// TIA Portal project "OPTS_scale_main_V1" (V16)

(* hardware
DEVICE "S71500/ET200MP station_1"  S7-1500 station
   slot 0: "Rail_0"  Rack  6ES7 590-1***0-0AA0
   slot 1: "PLC_1"  CPU 1516F-3 PN/DP  6ES7 516-3FN01-0AB0  V1.8
      slot 3: "CPU display_1"  6ES7591-1BA00-0AA0
      slot 32768: "PROFINET interface_1"  X1
         slot 32769: "Port_1"  X1 P1
         slot 32770: "Port_2"  X1 P2
      slot 33024: "PROFINET interface_2"  X2
         slot 33025: "Port_1"  X2 P1
      slot 33280: "DP interface_1"  X3
   slot 2: "DI 32x24VDC HF_1"  DI 32x24VDC HF  6ES7 521-1BL00-0AB0  V2.1
   slot 3: "DQ 32x24VDC/0.5A ST_1"  DQ 32x24VDC/0.5A ST  6ES7 522-1BL00-0AB0  V2.0
   slot 4: "AI 8xU/I/RTD/TC ST_1"  AI 8xU/I/RTD/TC ST  6ES7 531-7KF00-0AB0  V2.0
   slot 5: "AQ 4xU/I ST_1"  AQ 4xU/I ST  6ES7 532-5HD00-0AB0  V2.0
DEVICE "HMI_1"  HMI.Device
*)

// ===== PLC "PLC_1"  CPU 1516F-3 PN/DP =====

VAR_GLOBAL   // PLC tag table "OPTS_tag_table"
   "onOffSwitch" AT %I2.0 : Bool;
   "FL_PositionSensor" AT %IW138 : Int;
   "FR_PositionSensor" AT %IW140 : Int;
   "BL_PositionSensor" AT %IW132 : Int;
   "BR_PositionSensor" AT %IW130 : Int;
   "sensorXValue" AT %IW134 : Int;
   "sensorZValue" AT %IW136 : Int;
   "flOut" AT %QW4 : Int;
   "frOut" AT %QW6 : Int;
END_VAR

DATA_BLOCK "SensorProcessing_DB"   // DB1
{ S7_Optimized_Access := 'TRUE' }
VERSION : 0.1
// stored: InstanceOfName SensorProcessing
"SensorProcessing"
BEGIN
END_DATA_BLOCK

DATA_BLOCK "TargetInDistance_DB"   // DB2
{ S7_Optimized_Access := 'TRUE' }
VERSION : 0.1
// stored: InstanceOfName TargetInDistance
"TargetInDistance"
BEGIN
END_DATA_BLOCK

DATA_BLOCK "TargetInDistance_DB_1"   // DB3
{ S7_Optimized_Access := 'TRUE' }
VERSION : 0.1
// stored: InstanceOfName TargetInDistance
"TargetInDistance"
BEGIN
END_DATA_BLOCK

DATA_BLOCK "TargetInDistance_DB_2"   // DB4
{ S7_Optimized_Access := 'TRUE' }
VERSION : 0.1
// stored: InstanceOfName TargetInDistance
"TargetInDistance"
BEGIN
END_DATA_BLOCK

DATA_BLOCK "TargetInDistance_DB_3"   // DB5
{ S7_Optimized_Access := 'TRUE' }
VERSION : 0.1
// stored: InstanceOfName TargetInDistance
"TargetInDistance"
BEGIN
END_DATA_BLOCK

FUNCTION_BLOCK "SensorProcessing"   // FB1, FBD
{ S7_Optimized_Access := 'TRUE' }
VERSION : 0.1
   VAR_INPUT
      sensorX : Int;
      sensorZ : Int;
      scale : Real;
      pi : Real;
      edgeToMiddle : Real := 150.0;
   END_VAR
   VAR_OUTPUT
      LA_FL_Target : Real;
      LA_FR_Target : Real;
      LA_BL_Target : Real;
      LA_BR_Target : Real;
   END_VAR
   VAR
      xActuatorAdjustVolt : Real;
      zActuatorAdjustVolt : Real;
      xActuatorAdjustVoltInv : Real;
      zActuatorAdjustVoltInv : Real;
   END_VAR
   VAR_TEMP
      xAngle : Real;
      zAngle : Real;
      xAngleTangent : Real;
      zAngleTangent : Real;
      xActuatorAdjust : Real;
      zActuatorAdjust : Real;
      xActuatorAdjustNorm : Real;
      zActuatorAdjustNorm : Real;
   END_VAR
BEGIN

REGION Network 1
   // Converting sensor data for X axis to an angle in radian.
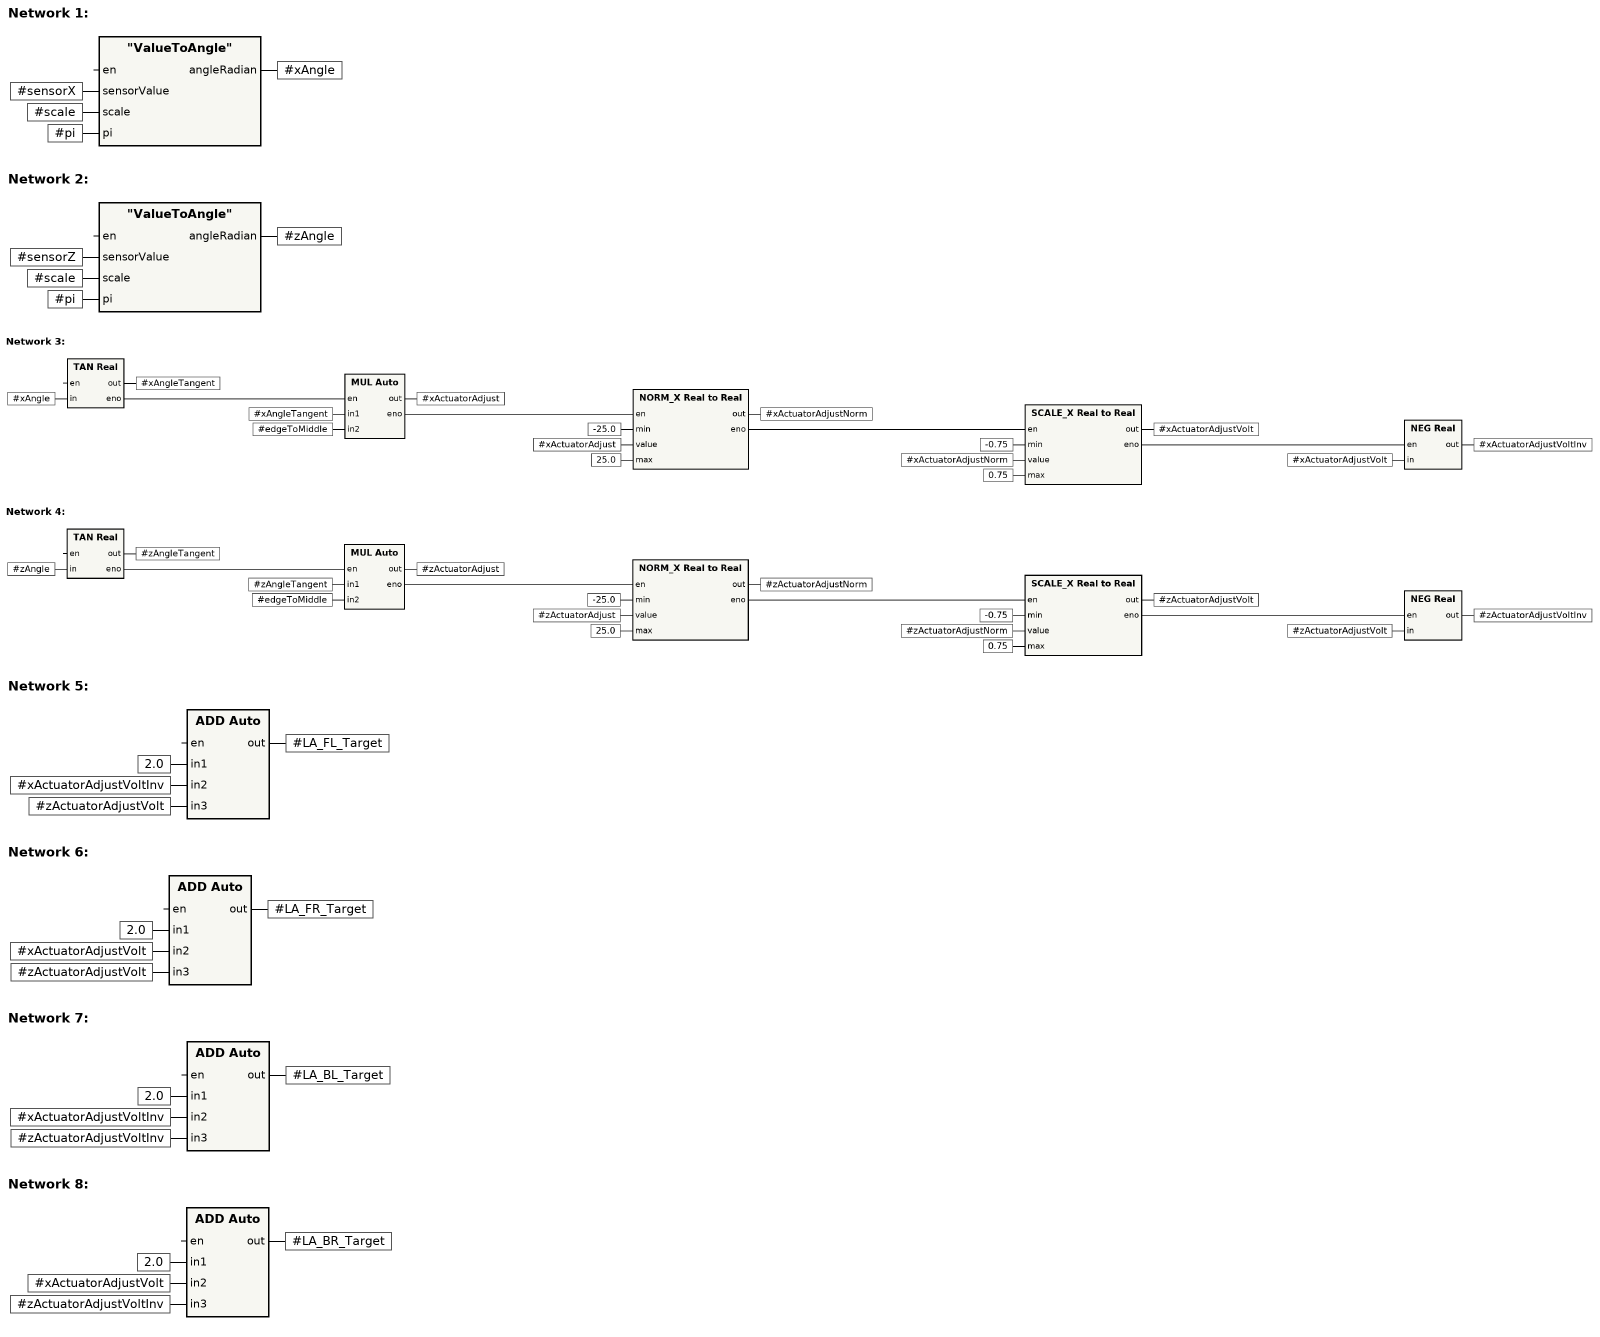
   "ValueToAngle"(sensorValue := #sensorX, scale := #scale, pi := #pi, angleRadian => #xAngle);
END_REGION

REGION Network 2
   // Converting sensor data for Z axis to an angle in radian.
   "ValueToAngle"(sensorValue := #sensorZ, scale := #scale, pi := #pi, angleRadian => #zAngle);
END_REGION

REGION Network 3
   // Calculating the distance the actuators have to be offset from the center for the X axis (left to right tilting)
   #xAngleTangent := TAN(#xAngle);
   #xActuatorAdjust := #xAngleTangent * #edgeToMiddle;
   #xActuatorAdjustNorm := NORM_X(MIN := -25.0, VALUE := #xActuatorAdjust, MAX := 25.0);
   #xActuatorAdjustVolt := SCALE_X(MIN := -0.75, VALUE := #xActuatorAdjustNorm, MAX := 0.75);
   #xActuatorAdjustVoltInv := -#xActuatorAdjustVolt;
END_REGION

REGION Network 4
   // Calculating the distance the actuators have to be offset from the center for the Z axis (front to back tilting)
   #zAngleTangent := TAN(#zAngle);
   #zActuatorAdjust := #zAngleTangent * #edgeToMiddle;
   #zActuatorAdjustNorm := NORM_X(MIN := -25.0, VALUE := #zActuatorAdjust, MAX := 25.0);
   #zActuatorAdjustVolt := SCALE_X(MIN := -0.75, VALUE := #zActuatorAdjustNorm, MAX := 0.75);
   #zActuatorAdjustVoltInv := -#zActuatorAdjustVolt;
END_REGION

REGION Network 5
   // Calculating target position for Front Left actuator, sum of adjustment in the X distance and Z distance, +2 for the center of the actuator.
   #LA_FL_Target := 2.0 + #xActuatorAdjustVoltInv + #zActuatorAdjustVolt;
END_REGION

REGION Network 6
   // Calculating target position for Front Right actuator, sum of adjustment in the X distance and Z distance, +2 for the center of the actuator.
   #LA_FR_Target := 2.0 + #xActuatorAdjustVolt + #zActuatorAdjustVolt;
END_REGION

REGION Network 7
   // Calculating target position for Rear Left actuator, sum of adjustment in the X distance and Z distance, +2 for the center of the actuator.
   #LA_BL_Target := 2.0 + #xActuatorAdjustVoltInv + #zActuatorAdjustVoltInv;
END_REGION

REGION Network 8
   // Calculating target position for Rear Right actuator, sum of adjustment in the X distance and Z distance, +2 for the center of the actuator.
   #LA_BR_Target := 2.0 + #xActuatorAdjustVolt + #zActuatorAdjustVoltInv;
END_REGION
END_FUNCTION_BLOCK

FUNCTION_BLOCK "TargetInDistance"   // FB3, FBD
{ S7_Optimized_Access := 'TRUE' }
VERSION : 0.1
   VAR_INPUT
      targetVoltage : Real;
   END_VAR
   VAR_OUTPUT
      targetDistance : Real;
   END_VAR
   VAR_TEMP
      help : Real;
   END_VAR
BEGIN

REGION Network 1
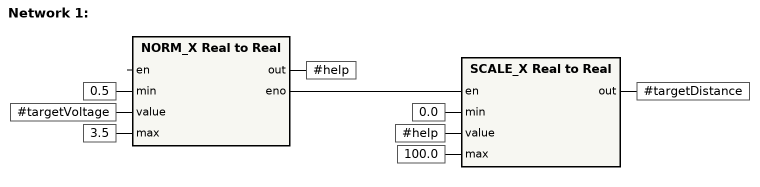
   #help := NORM_X(MIN := 0.5, VALUE := #targetVoltage, MAX := 3.5);
   #targetDistance := SCALE_X(MIN := 0.0, VALUE := #help, MAX := 100.0);
END_REGION
END_FUNCTION_BLOCK

FUNCTION "ValueToAngle" : Void   // FC1, FBD
{ S7_Optimized_Access := 'TRUE' }
VERSION : 0.1
   VAR_INPUT
      sensorValue : Int;
      scale : Real;
      pi : Real;
   END_VAR
   VAR_OUTPUT
      angleRadian : Real;
   END_VAR
   VAR_TEMP
      sensorValueReal : Real;
      sensorValueNorm : Real;
      angleDegree : Real;
      angleHelpValue : Real;
   END_VAR
BEGIN

REGION Network 1
   // This network converts the sensorValue from an Int to a Real datatype.
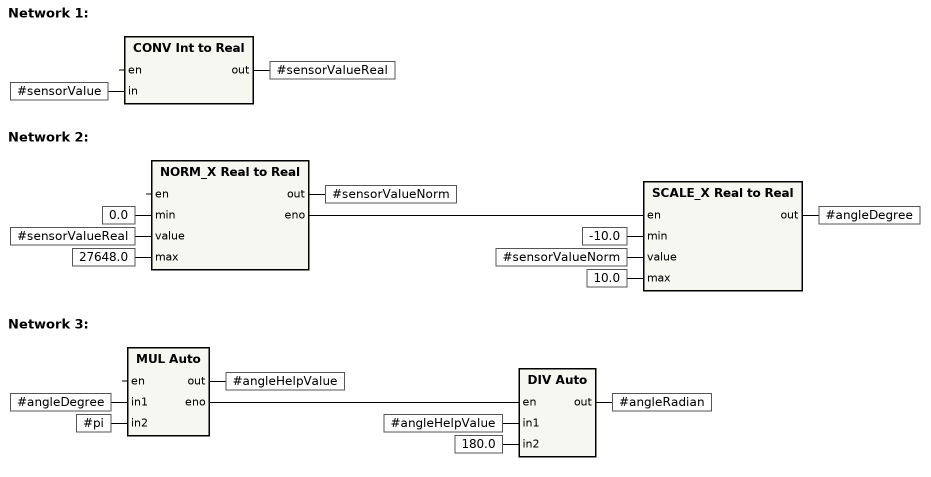
   #sensorValueReal := INT_TO_REAL(#sensorValue);
END_REGION

REGION Network 2
   // Convert the data from very high number to an angle.
   #sensorValueNorm := NORM_X(MIN := 0.0, VALUE := #sensorValueReal, MAX := 27648.0);
   #angleDegree := SCALE_X(MIN := -10.0, VALUE := #sensorValueNorm, MAX := 10.0);
END_REGION

REGION Network 3
   // Convert degrees to radian
   #angleHelpValue := #angleDegree * #pi;
   #angleRadian := #angleHelpValue / 180.0;
END_REGION
END_FUNCTION

ORGANIZATION_BLOCK "Main"   // OB1, FBD, ProgramCycle
TITLE = "Main Program Sweep (Cycle)"
{ S7_Optimized_Access := 'TRUE' }
VERSION : 0.1
   VAR_INPUT
      Initial_Call : Bool;   // Initial call of this OB
      Remanence : Bool;   // =True, if remanent data are available
   END_VAR
   VAR_TEMP
      flInTemp : Real;
      frInTemp : Real;
      blInTemp : Real;
      brInTemp : Real;
   END_VAR
BEGIN

REGION Network 1
   // Get positions for the linear actuators
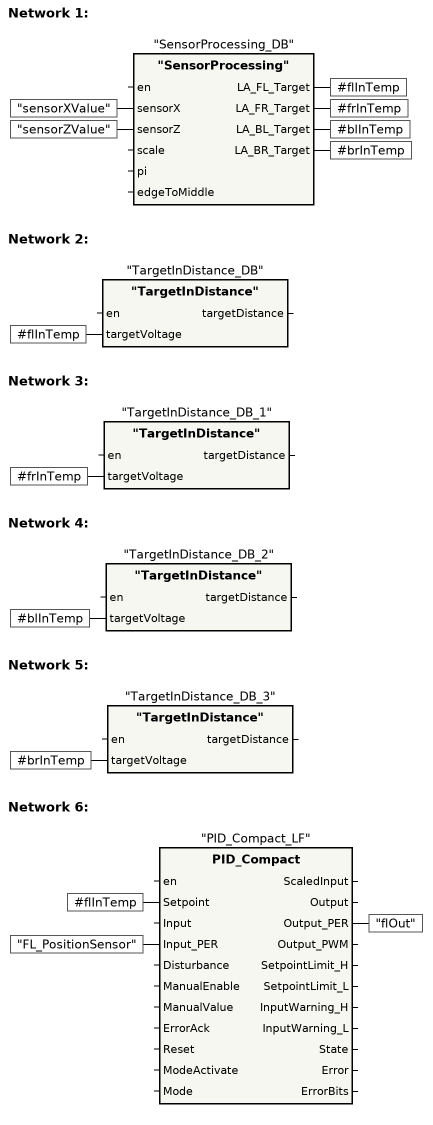
   "SensorProcessing_DB"(sensorX := "sensorXValue",   // "SensorProcessing"
                         sensorZ := "sensorZValue",
                         LA_FL_Target => #flInTemp,
                         LA_FR_Target => #frInTemp,
                         LA_BL_Target => #blInTemp,
                         LA_BR_Target => #brInTemp);
END_REGION

REGION Network 2
   "TargetInDistance_DB"(targetVoltage := #flInTemp);   // "TargetInDistance"
END_REGION

REGION Network 3
   "TargetInDistance_DB_1"(targetVoltage := #frInTemp);   // "TargetInDistance"
END_REGION

REGION Network 4
   "TargetInDistance_DB_2"(targetVoltage := #blInTemp);   // "TargetInDistance"
END_REGION

REGION Network 5
   "TargetInDistance_DB_3"(targetVoltage := #brInTemp);   // "TargetInDistance"
END_REGION

REGION Network 6
   "PID_Compact_LF"(Setpoint := #flInTemp, Input_PER := "FL_PositionSensor", Output_PER => "flOut");   // PID_Compact
END_REGION
END_ORGANIZATION_BLOCK

ORGANIZATION_BLOCK "Startup"   // OB100, FBD, Startup
TITLE = "Complete Restart"
{ S7_Optimized_Access := 'TRUE' }
VERSION : 0.1
   VAR_INPUT
      LostRetentive : Bool;   // True if retentive data are lost
      LostRTC : Bool;   // True if date and time are lost
   END_VAR
BEGIN

REGION Network 1
   // Calculate pi value for later use.
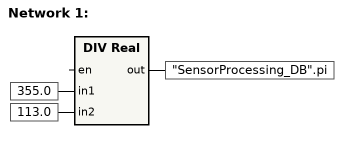
   "SensorProcessing_DB".pi := 355.0 / 113.0;
END_REGION
END_ORGANIZATION_BLOCK